FUNCTION_BLOCK PrintStation EXTENDS MachineStation
VAR_INPUT
	rIO				: REFERENCE TO Print_IO_typ;
	rMultiStn		: REFERENCE TO MultiStation;
	rVisionStation	: REFERENCE TO Station;
END_VAR
VAR_OUTPUT
END_VAR
VAR
Payload	: Payload_typ;
	i: INT;
END_VAR

(*IF rStation = 0 OR rIO = 0 THEN		HOW DO I CHECK FOR THIS???
	RETURN;
END_IF	*)

// Catch Incoming Shuttles and assign to station
IF rMultiStn.PositionTrigger.MoverPassedPosition THEN
	rMultiStn.PosTriggerPayload	:= rMultiStn.PositionTrigger.CurrentMover.Payload;
	// TODO add check for Payload info to reject ball or another reason we wouldnt want to print
	rMultiStn.PositionTrigger.CurrentMover.MoveToStation(rMultiStn.Station[0]);
	rMultiStn.PositionTrigger.MuteCurrent();
END_IF

// Station Sequence
IF Enable THEN
	IF NOT _Enable THEN
		;
	END_IF

	CASE State OF
		STN_WAIT:
			IF rMultiStn.AllMoversInPosition THEN
				FOR i := 0 TO GVL.MULTISTN_NUM_STN - 1 DO
					IF rMultiStn.Station[i].TrackedMoverCount > 0 THEN
						rMultiStn.StationPayload[i]	:= rMultiStn.Station[i].CurrentMover.Payload;
					END_IF
				END_FOR
				Payload				:= rMultiStn.CurrentMover.Payload;
				rIO.Outputs.Print	:= TRUE;
				State				:= STN_PROCESS;
			END_IF

		STN_PROCESS:
			IF rIO.Inputs.PrintComplete THEN
				rIO.Outputs.Print		:= FALSE;
				FOR i := 0 TO GVL.MULTISTN_NUM_STN - 1 DO
					IF rMultiStn.Station[i].TrackedMoverCount > 0 THEN
						rMultiStn.StationPayload[i].PrintStepComplete[i]	:= TRUE;
						IF i = 3 THEN
							rMultiStn.StationPayload[i].PrintComplete		:= TRUE;
						END_IF
					END_IF
				END_FOR
			State						:= STN_SEND;
			END_IF

		STN_SEND:
			// Write Payload Data
			FOR i := 0 TO GVL.MULTISTN_NUM_STN - 1 DO
				IF rMultiStn.Station[i].TrackedMoverCount > 0 THEN
					rMultiStn.Station[i].CurrentMover.Payload	:= rMultiStn.StationPayload[i];
				END_IF
			END_FOR

			// Send Mover
			FOR i := 3 TO 0 BY -1 DO
				IF rMultiStn.Station[i].TrackedMoverCount > 0 THEN
					IF i = 3 THEN
						rMultiStn.Station[i].CurrentMover.MoveToStation(rVisionStation);
					ELSE
						rMultiStn.Station[i].CurrentMover.MoveToStation(rMultiStn.Station[i+1]);
					END_IF
				END_IF
				IF i = 0 THEN EXIT; END_IF
			END_FOR
			State		:= STN_WAIT;
		
		STN_ERROR:
	
	END_CASE

ELSIF _Enable THEN
	;
END_IF

//Save Previous Values
_Enable	:= Enable;

METHOD Cyclic : BOOL
VAR_INPUT
END_VAR
END_METHOD

END_FUNCTION_BLOCK

(* stored: Version 1.1.0.1, ProductVersion 3.1.4024.12
   POU PrintStation: Id {bbe07669-1b09-0bc2-0cf7-35c98289024b}, SpecialFunc None
   Method Cyclic: Id {06adf546-a0d7-0c76-24f1-705bd756794d} *)
